SUBAPPLICATION Uebung_012o_AR2 (* VT-Feld UND OPC-UA (letzter Schreiber gewinnt) und Speichern INI via AR2 - NumericValue_TO_AR2_OPC direkt an ein INI_AR2 angeschlossen *)
  (* Standard: 61499-2; Description: Copyright (c) 2026 Meisterschulen am Ostbahnhof This program and the accompanying materials are made available under the terms of the Eclipse Public License 2.0 which is available at https://www.eclipse.org/legal/epl-2.0/ SPDX-License-Identifier: EPL-2.0 *)
  (* Version 1.0, 2026-08-31, Franz Höpfinger, Meisterschulen am Ostbahnhof, VT+OPC sibling of Uebung_012g_AR2 (VT only) / Uebung_012i_AR2 (OPC only) - NumericValue_TO_AR2_OPC direkt an INI_AR2 *)
  PACKAGE Uebungen;
  IMPORT Uebungen::const::NVS::NVS_Keys::KEY_I1_STORE;
  IMPORT Uebungen::const::NVS::NVS_Keys::SECTION_I1_STORE;
  IMPORT Uebungen::const::UT::DefaultPool_Numeric::InputNumber_I1_N;
  IMPORT Uebungen::const::OPC::OPC_Strings::Uebung12o_READ;
  IMPORT Uebungen::const::OPC::OPC_Strings::Uebung12o_WRITE;
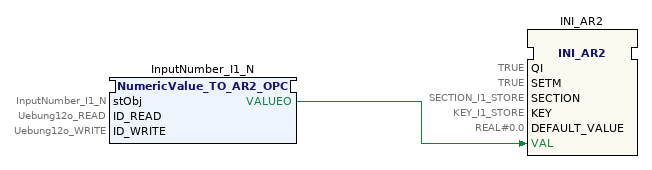
  (* SETM=TRUE ist hier ESSENTIELL (anders als bei den reinen VT- oder OPC-Uebungen): es gibt ZWEI Quellen (VT + Remote). Aendert der Operator den Wert am VT-Feld, muss die Remote-Seite das sofort mitbekommen (Publish-Echo) - und umgekehrt. Ohne SETM=TRUE wuerde die jeweils andere Seite von einer Live-Aenderung nichts erfahren, erst der naechste Neustart wuerde sie synchronisieren. *)
  FBS
    INI_AR2 : eclipse4diac::storage::INI_AR2(QI := TRUE, SETM := TRUE, SECTION := SECTION_I1_STORE, KEY := KEY_I1_STORE, DEFAULT_VALUE := REAL#0.0);
  END_FBS
  SUBAPPS
    InputNumber_I1_N : MyLib::sys::NumericValue_TO_AR2_OPC(stObj := InputNumber_I1_N, ID_READ := Uebung12o_READ, ID_WRITE := Uebung12o_WRITE);
  END_SUBAPPS
  ADAPTER_CONNECTIONS
    InputNumber_I1_N.VALUEO TO INI_AR2.VAL;
  END_CONNECTIONS
END_SUBAPPLICATION
